// TIA Portal V21 export
FUNCTION "GestPid_Comando1Valvola" : Void   // FC66, LAD
{ S7_Optimized_Access := 'TRUE' }
// stored: SetENOAutomatically false
   VAR_INPUT
      K_Valvola : Int;
      K_Pid : Int;
      K_TipoOutValvola : Int;
   END_VAR
BEGIN

REGION Network 1 (SCL)
   "Pid".P[#K_Pid].In.K_Valvola1 := #K_Valvola;
   IF #K_TipoOutValvola = "K_TipoOutValvola_Portata" THEN
       "Valvola".V[#K_Valvola].Hmi.Visibilita.ModulantePortata := True;
   END_IF;
   IF #K_TipoOutValvola = "K_TipoOutValvola_Pressione" THEN
       "Valvola".V[#K_Valvola].Hmi.Visibilita.ModulantePressione := True;
   END_IF;
END_REGION
END_FUNCTION
